TEXTLIST OriConvention
  0 = 'ADDAXES'
  1 = 'ZYZ'
  2 = 'ZYX'
  3 = 'XYZ'
   = ''
END_TEXTLIST

(* stored: Version 1.1.0.1
   TextList OriConvention: Id {1953da2c-4f47-4be6-9946-cd85868dd801} *)
